// TIA Portal V21 export
FUNCTION_BLOCK "FB102"   // FB102, LAD
TITLE = FB102
{ S7_Optimized_Access := 'FALSE' }
AUTHOR : PRECISE
FAMILY : PRECISE
// On Off Delay
// stored: AutoNumber false, SetENOAutomatically false
   VAR_INPUT
      Enable : Bool;
      Running : Bool;
      SecPulse : Bool;
      OnTimeSV : Int := 3;
      OffTimeSV : Int := 3;
   END_VAR
   VAR_OUTPUT
      Valve : Bool;
   END_VAR
   VAR_IN_OUT
      ValveBit : Bool;
      RE : Bool;
      OnTimePV : Int;
      OffTimePV : Int;
   END_VAR
   VAR_TEMP   // added for the SCL form of the ladder/FBD networks
      _w1 : Bool;
      _w2 : Bool;
      _w3 : Bool;
   END_VAR
BEGIN

REGION Network 1: Start
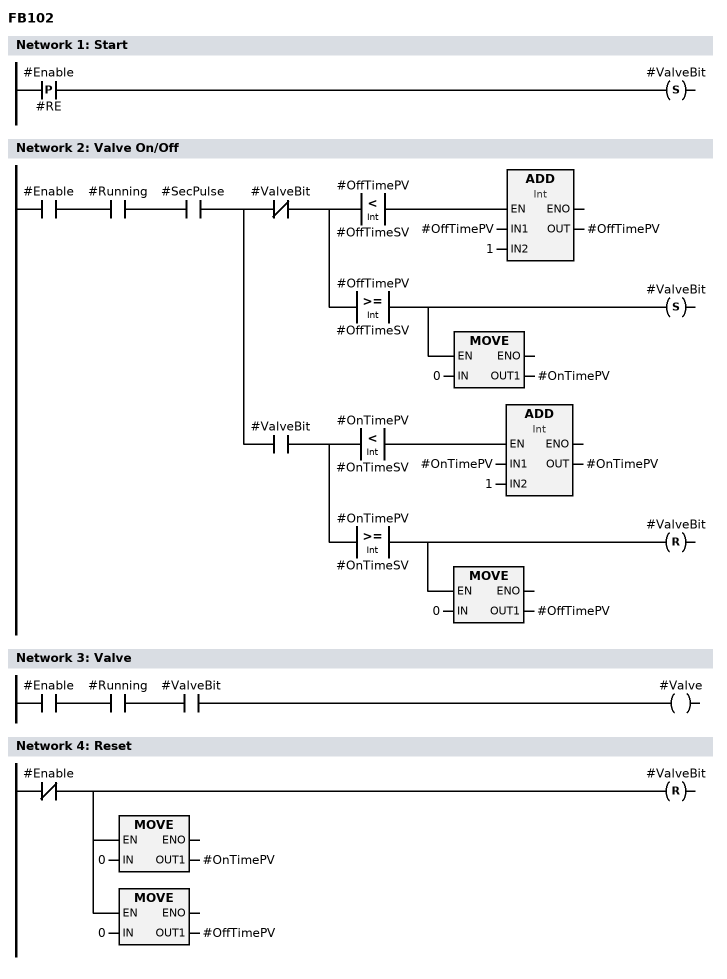
   RUNG wire#powerrail
      P_Contact(operand := #Enable, bit := #RE)
      S_Coil( #ValveBit )
   END_RUNG
   // the same network as SCL:
   #_w1 := #Enable AND NOT #RE;   // rising edge of #Enable
   #RE := #Enable;
   IF #_w1 THEN #ValveBit := TRUE; END_IF;
END_REGION

REGION Network 2: Valve On/Off
   RUNG wire#powerrail
      Contact( #Enable )
      Contact( #Running )
      Contact( #SecPulse )
      wire#w1
      I_Contact( #ValveBit )
      wire#w2
      { S7_Templates := "SrcType := Int" } LT_Contact(in1 := #OffTimePV, in2 := #OffTimeSV)
      { S7_Templates := "SrcType := Int"; S7_GenerateENO := "TRUE" } Add(in1 := #OffTimePV, in2 := 1, out => #OffTimePV)
   END_RUNG
   RUNG wire#w2
      { S7_Templates := "SrcType := Int" } GE_Contact(in1 := #OffTimePV, in2 := #OffTimeSV)
      wire#w3
      S_Coil( #ValveBit )
   END_RUNG
   RUNG wire#w3
      { S7_GenerateENO := "TRUE" } Move(in := 0, out1 => #OnTimePV)
   END_RUNG
   RUNG wire#w1
      Contact( #ValveBit )
      wire#w4
      { S7_Templates := "SrcType := Int" } LT_Contact(in1 := #OnTimePV, in2 := #OnTimeSV)
      { S7_Templates := "SrcType := Int"; S7_GenerateENO := "TRUE" } Add(in1 := #OnTimePV, in2 := 1, out => #OnTimePV)
   END_RUNG
   RUNG wire#w4
      { S7_Templates := "SrcType := Int" } GE_Contact(in1 := #OnTimePV, in2 := #OnTimeSV)
      wire#w5
      R_Coil( #ValveBit )
   END_RUNG
   RUNG wire#w5
      { S7_GenerateENO := "TRUE" } Move(in := 0, out1 => #OffTimePV)
   END_RUNG
   // the same network as SCL:
   #_w1 := #Enable AND #Running AND #SecPulse;
   #_w2 := #_w1 AND NOT #ValveBit;
   IF #_w2 AND (#OffTimePV < #OffTimeSV) THEN #OffTimePV := #OffTimePV + 1; END_IF;
   IF #_w2 AND (#OffTimePV >= #OffTimeSV) THEN
       #ValveBit := TRUE;
       #OnTimePV := 0;
   END_IF;
   #_w3 := #_w1 AND #ValveBit;
   IF #_w3 AND (#OnTimePV < #OnTimeSV) THEN #OnTimePV := #OnTimePV + 1; END_IF;
   IF #_w3 AND (#OnTimePV >= #OnTimeSV) THEN
       #ValveBit := FALSE;
       #OffTimePV := 0;
   END_IF;
END_REGION

REGION Network 3: Valve
   RUNG wire#powerrail
      Contact( #Enable )
      Contact( #Running )
      Contact( #ValveBit )
      Coil( #Valve )
   END_RUNG
   // the same network as SCL:
   #Valve := #Enable AND #Running AND #ValveBit;
END_REGION

REGION Network 4: Reset
   RUNG wire#powerrail
      I_Contact( #Enable )
      wire#w1
      R_Coil( #ValveBit )
   END_RUNG
   RUNG wire#w1
      { S7_GenerateENO := "TRUE" } Move(in := 0, out1 => #OnTimePV)
   END_RUNG
   RUNG wire#w1
      { S7_GenerateENO := "TRUE" } Move(in := 0, out1 => #OffTimePV)
   END_RUNG
   // the same network as SCL:
   IF NOT #Enable THEN
       #ValveBit := FALSE;
       #OnTimePV := 0;
       #OffTimePV := 0;
   END_IF;
END_REGION
END_FUNCTION_BLOCK
